(* Logix 5000 project; controller Lab4_main vendor 1 type 14 code 3 rev 13.31; software revision 13.03 *)
// EE: Angelino Lefevers
// Lab 4 main program

TASK MainTask (continuous, watchdog 500 ms) : MainProgram

MODULES
   Local : vendor 1 type 14 code 3 (ICP 0, rev 13.31)
      Digital_IN : 1756-IB16 (ICP 2, rev 2.1, Input RPI 10 ms)
      Digital_OUT : vendor 1 type 7 code 18 (ICP 4, rev 1.1, Output RPI 10 ms)
      Analog_IN : 1756-IF8 (ICP 6, rev 1.1, Input RPI 100 ms)
      Analog_OUT : 1756-OF4 (ICP 7, rev 1.1, Output RPI 12 ms)
END_MODULES

PROGRAM MainProgram   (* routine attr 65 MainRoutine *)

ROUTINE MainRoutine   (* ladder *)
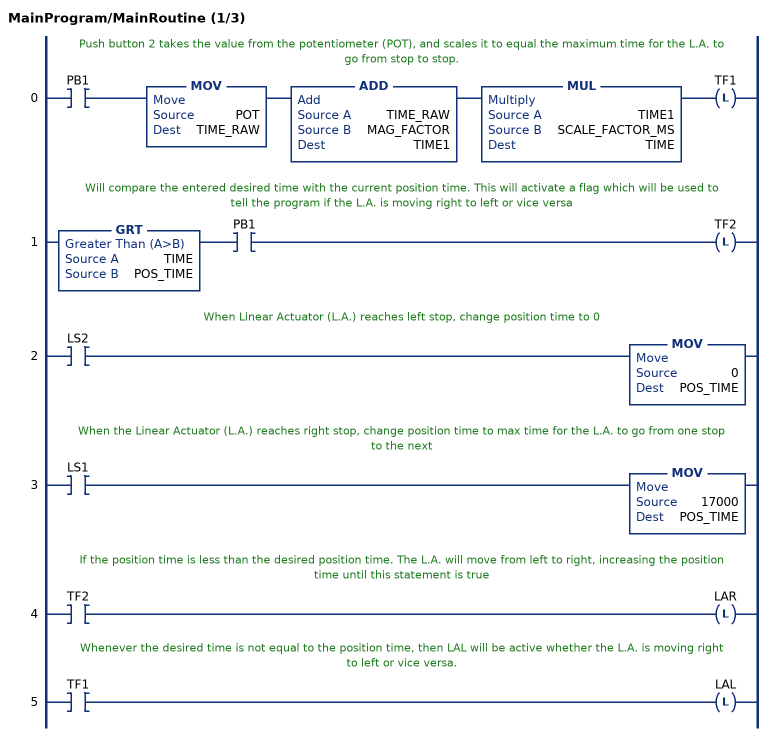
   // Push button 2 takes the value from the potentiometer (POT), and scales it to equal the maximum time for the L.A. to go from stop to stop.
   0: XIC(PB1)MOV(POT,TIME_RAW)ADD(TIME_RAW,MAG_FACTOR,TIME1)MUL(TIME1,SCALE_FACTOR_MS,TIME)OTL(TF1);
   // Will compare the entered desired time with the current position time. This will activate a flag which will be used to tell the program if the L.A. is moving right to left or vice versa
   1: GRT(TIME,POS_TIME)XIC(PB1)OTL(TF2);
   // When Linear Actuator (L.A.) reaches left stop, change position time to 0
   2: XIC(LS2)MOV(0,POS_TIME);
   // When the Linear Actuator (L.A.) reaches right stop, change position time to max time for the L.A. to go from one stop to the next
   3: XIC(LS1)MOV(17000,POS_TIME);
   // If the position time is less than the desired position time. The L.A. will move from left to right, increasing the position time until this statement is true
   4: XIC(TF2)OTL(LAR);
   // Whenever the desired time is not equal to the position time, then LAL will be active whether the L.A. is moving right to left or vice versa.
   5: XIC(TF1)OTL(LAL);
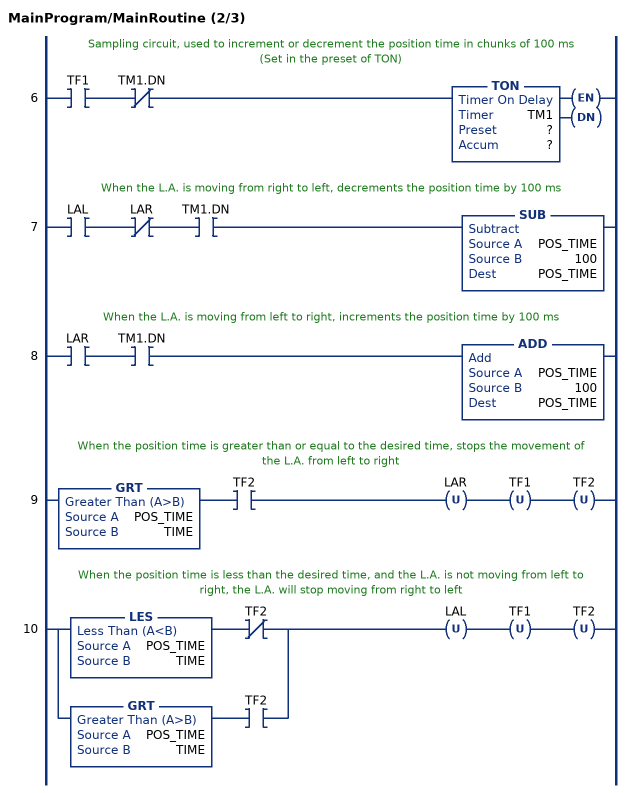
   // Sampling circuit, used to increment or decrement the position time in chunks of 100 ms (Set in the preset of TON)
   6: XIC(TF1)XIO(TM1.DN)TON(TM1,?,?);
   // When the L.A. is moving from right to left, decrements the position time by 100 ms
   7: XIC(LAL)XIO(LAR)XIC(TM1.DN)SUB(POS_TIME,100,POS_TIME);
   // When the L.A. is moving from left to right, increments the position time by 100 ms
   8: XIC(LAR)XIC(TM1.DN)ADD(POS_TIME,100,POS_TIME);
   // When the position time is greater than or equal to the desired time, stops the movement of the L.A. from left to right
   9: GRT(POS_TIME,TIME)XIC(TF2)OTU(LAR)OTU(TF1)OTU(TF2);
   // When the position time is less than the desired time, and the L.A. is not moving from left to right, the L.A. will stop moving from right to left
   10: [LES(POS_TIME,TIME) XIO(TF2) ,GRT(POS_TIME,TIME) XIC(TF2) ]OTU(LAL)OTU(TF1)OTU(TF2);
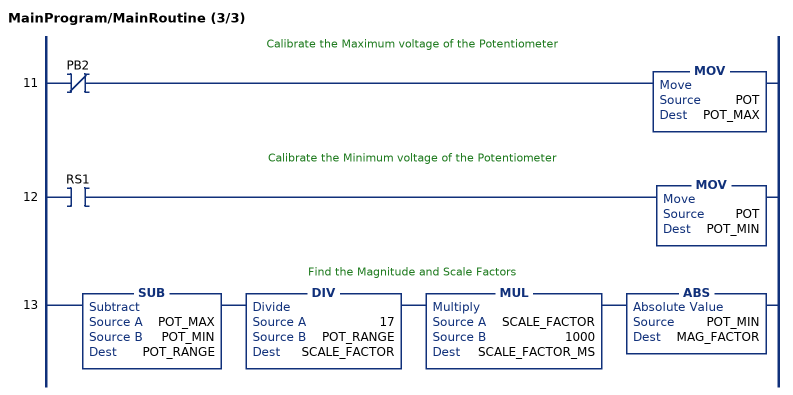
   // Calibrate the Maximum voltage of the Potentiometer
   11: XIO(PB2)MOV(POT,POT_MAX);
   // Calibrate the Minimum voltage of the Potentiometer
   12: XIC(RS1)MOV(POT,POT_MIN);
   // Find the Magnitude and Scale Factors
   13: SUB(POT_MAX,POT_MIN,POT_RANGE)DIV(17,POT_RANGE,SCALE_FACTOR)MUL(SCALE_FACTOR,1000,SCALE_FACTOR_MS)ABS(POT_MIN,MAG_FACTOR);
END_ROUTINE
END_PROGRAM
